{attribute 'no_explicit_call' := 'Do not call the body - Stick to OOP'}
FUNCTION_BLOCK FB_CoE_UINT EXTENDS FB_CoE_Base
(* 
   FB_init:
	(	ipCoeConnection := fbCoeConnection, (*each EC-Slave needs one FB_CoE_Connection*)
		nIndex     		:= 16#8010, (* CoE Object Index *)
		nSubIndex  		:= 16#11 (* Subindex of CoE Object *));
 *)
VAR
	{attribute 'hide'}
	nValue : UINT;
END_VAR

PROPERTY PROTECTED cbBufLen : UDINT
GET
cbBufLen := SIZEOF(nValue);
END_GET
END_PROPERTY

PROPERTY PROTECTED pSrcBuf : PVOID
GET
pSrcBuf := ADR(nValue);
END_GET
END_PROPERTY

{attribute 'monitoring':='call'}
PROPERTY Value : UINT
GET
Value := nValue;
END_GET
SET
nValue := Value;

//Trigger a new write cycle
THIS^.bWriteDone 	:= FALSE;
END_SET
END_PROPERTY

END_FUNCTION_BLOCK

(* stored: Version 1.1.0.1, ProductVersion 3.1.4024.12
   POU FB_CoE_UINT: Id {c27c62dd-3346-46fc-9883-0e031ca0a44d}, SpecialFunc None
   Property cbBufLen: Id {416f0dc3-b439-4928-aa9a-9b8428e7bbd5}
   Get Get: Id {5d909c92-6645-44c2-b650-2d490bf1f390}
   Property pSrcBuf: Id {bf987af5-d941-4559-888b-3f709f3f8146}
   Get Get: Id {ca7e6833-baf3-4ad8-a76f-f3b779e8dd3a}
   Property Value: Id {1fc2bfab-3af1-44c2-9a91-755340384697}
   Get Get: Id {ceaaf1da-d6be-402a-b354-8223d0807707}
   Set Set: Id {d992b438-4849-4d9b-b7e8-1c6dcc197b2e} *)
